// TIA Portal V18 export
TYPE "ST_GeneralAnalog"
   STRUCT
      Common : Struct   // 通用变量
         nMode : Int;   // 控制模式
         bEnable : Bool;   // 启动条件
         bError : Bool;   // 错误
         bWarning : Bool;   // 警告
         bReset : Bool;   // 复位
         bDone : Bool;   // 执行动作完成
         bScreenActive : Bool;   // 激活屏幕
         nErrorNo : Int;   // 错误代码
         nWarningNo : Int;   // 警告代码
         nLastStep : Int;   // 上一步号
         nCurrentStep : Int;   // 当前步号
         nNextStep : Int;   // 下一步号
         tMaxProcessTime : Time;   // 最大执行时间
         tActProcessTime : Time;   // 实际流程时间
      END_STRUCT;
      In : Struct   // PLC输入变量
         nActualValueX : UInt;   // 实际输入值
      END_STRUCT;
      Out : Struct   // PLC输出变量
         bReserved : Bool;   // 备用
      END_STRUCT;
      Para : Struct   // 参数变量
         General : Struct   // 通用变量
            rActualValueY : Real;   // 实时输出值
            rSlope : Real;   // 方程式斜率
            rConstant : Real;   // 方程式常数
            aPos : Array[1..2] of Struct   // 校准
               nValueX : UInt;   // 校准X
               nValueY : Real;   // 校准Y
            END_STRUCT;
         END_STRUCT;
         Set : Struct   // 参数设定
            rLimitMin : Real;   // 最小值
            rLimitMax : Real;   // 最大值
            aLimit : Array[0..9] of Struct   // 上下限
               rMin : Real;   // 下限
               rMax : Real;   // 上限
            END_STRUCT;
            nUnitX : Int;   // 输入单位
            nUnitY : Int;   // 输出单位
         END_STRUCT;
         Result : Struct   // 运算结果
            bOk : Bool;   // 结果OK
            bNok : Bool;   // 结果NG
            bOverMin : Bool;   // 超出下限值
            bOverMax : Bool;   // 超出上限值
            rValueY : Real;   // 测量结果输出值
         END_STRUCT;
         Record : Struct   // 数据记录
            bClear : Bool;   // 清除记录数据
            nSetNumber : Int;   // 设定记录个数
            nActNumber { ExternalVisible := 'False'} : Int;   // 显示记录到第几位
            rAverageValueY : Real;   // 平均值
            aValueY : Array[1..50] of Real;   // 记录值
         END_STRUCT;
      END_STRUCT;
   END_STRUCT;
END_TYPE
